// TIA Portal V18 export
// export: Created 2026-06-06T00:00:00Z, ExportSetting WithDefaults
DATA_BLOCK "{{DB_NAME}}"   // DB{{DB_NUMBER}}
TITLE = {{DB_NAME}}
{ S7_Optimized_Access := 'FALSE' }
VERSION : 0.1
// DB communication via Modbus TCP
// stored: AutoNumber false, IsOnlyStoredInLoadMemory false, IsWriteProtectedInAS false
   VAR
      MB_TCP : TCON_IP_v4;
   END_VAR
BEGIN
END_DATA_BLOCK
